{attribute 'linkalways'} 
{attribute 'no_explicit_call' := 'This FB is a CLASS and must be accessed using methods or properties'}
{attribute 'enable_dynamic_creation'}
FUNCTION_BLOCK FINAL GE_INT EXTENDS Node
VAR
	in1 : _INT(0);
	in2 : _INT(0);
	out : _BOOL(FALSE);
END_VAR

METHOD PUBLIC Clone : I_Node
VAR
	pNode : POINTER TO GE_INT;
END_VAR
pNode := __NEW(GE_INT);
Clone := pNode^;
END_METHOD

METHOD FB_init : BOOL
VAR_INPUT
	bInitRetains : BOOL; // if TRUE, the retain variables are initialized (warm start / cold start)
	bInCopyCode : BOOL;  // if TRUE, the instance afterwards gets moved into the copy code (online change)
END_VAR
AddInput('in1',THIS^.in1);
AddInput('in2',THIS^.in2);
AddOutput('out', THIS^.out);
END_METHOD

METHOD PROTECTED OnExecute
VAR
END_VAR
out.Value := in1.Value >= in2.Value;
END_METHOD

END_FUNCTION_BLOCK

(* stored: Version 1.1.0.1, ProductVersion 3.1.4024.15
   POU GE_INT: Id {be5f8b61-50ef-40e9-9c1a-c16e73aa7ab7}, SpecialFunc None
   Folder Constructor: Id {da177a02-9d8a-4d94-86b4-aa77bb9b1da0}
   Method Clone: Id {1cfd20dc-b00f-4eca-b5df-79dd4902ac4b}
   Method FB_init: Id {0b6da3a6-c397-4d51-bb79-0f4bd470ba86}
   Method OnExecute: Id {33fb7d82-42b8-4a50-987e-1b39b0cf9b79} *)
